FUNCTION_BLOCK ArrayCumulativeSquared (* Basic FB with empty ECC *)
  (* Standard: 61499-2; Function: Squaring each of numbers and sum it all; Description: Total of Square Array *)
  (* Version 1.0, 2020-07-18, CandraWardaya, UGM *)
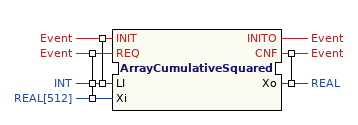
  EVENT_INPUT
    INIT WITH LI; (* Sending Array length Trigger *)
    REQ WITH Xi, LI; (* Request of Execution *)
  END_EVENT
  EVENT_OUTPUT
    INITO; (* Sending event for Setting Array length *)
    CNF WITH Xo; (* Confirmation of Execution *)
  END_EVENT
  VAR_INPUT
    LI : INT; (* Array Length *)
    Xi : ARRAY [0..511] OF REAL; (* Input real array *)
  END_VAR
  VAR_OUTPUT
    Xo : REAL; (* Output real, sum of component square array *)
  END_VAR
  VAR
    i : INT; (* Internal Variable *)
    X : REAL; (* Internal Variable *)
    val : REAL; (* Internal Variable *)
  END_VAR
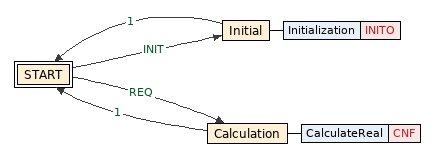
  EC_STATES
    START; (* Initial State *)
    Calculation : CalculateReal -> CNF;
    Initial : Initialization -> INITO;
  END_STATES
  EC_TRANSITIONS
    Calculation TO START := 1;
    START TO Initial := INIT;
    Initial TO START := 1;
    START TO Calculation := REQ;
  END_TRANSITIONS
  ALGORITHM CalculateReal IN ST: (* New Algorithm *)
val :=0;
for i:=0 to LI-1 do
	val := val + EXPT(Xi[i],2);
end_for;
Xo := val;
  END_ALGORITHM
  ALGORITHM Initialization IN ST: (* New Algorithm *)

  END_ALGORITHM
END_FUNCTION_BLOCK
